# EPICS autosave request: mrfApp/Db/evr-template-pulse-gen-generic.inc.req
$(P)$(R)PulseGen@PULSE_GEN_NUM@:Enabled.VAL
$(P)$(R)PulseGen@PULSE_GEN_NUM@:MapResetEnabled.VAL
$(P)$(R)PulseGen@PULSE_GEN_NUM@:MapSetEnabled.VAL
$(P)$(R)PulseGen@PULSE_GEN_NUM@:MapTrigEnabled.VAL
$(P)$(R)PulseGen@PULSE_GEN_NUM@:Polarity.VAL
